{attribute 'qualified_only'}
VAR_GLOBAL CONSTANT
	strExportDirectory : STRING := 'C:\testresult\';
END_VAR

(* stored: Version 1.1.0.1, ProductVersion 3.1.4024.13
   GVL GVL_Parameter: Id {06b1eece-8629-4f9e-b6a4-2d2d8f628d63}, ParameterList True *)
